{attribute 'linkalways'} 
{attribute 'no_explicit_call' := 'This FB is a CLASS and must be accessed using methods or properties'}
{attribute 'enable_dynamic_creation'}
FUNCTION_BLOCK FINAL MIN_LWORD EXTENDS Node
VAR
	in1 : _LWORD(0);
	in2 : _LWORD(0);
	out : _LWORD(0);
END_VAR

METHOD PUBLIC Clone : I_Node
VAR
	pNode : POINTER TO MIN_LWORD;
END_VAR
pNode := __NEW(MIN_LWORD);
Clone := pNode^;
END_METHOD

METHOD FB_init : BOOL
VAR_INPUT
	bInitRetains : BOOL; // if TRUE, the retain variables are initialized (warm start / cold start)
	bInCopyCode : BOOL;  // if TRUE, the instance afterwards gets moved into the copy code (online change)
END_VAR
AddInput('in1',THIS^.in1);
AddInput('in2',THIS^.in2);
AddOutput('out', THIS^.out);
END_METHOD

METHOD PROTECTED OnExecute
VAR
END_VAR
out.Value := MIN(in1.Value, in2.Value);
END_METHOD

END_FUNCTION_BLOCK

(* stored: Version 1.1.0.1, ProductVersion 3.1.4024.15
   POU MIN_LWORD: Id {a3934d77-3451-408a-9885-6d7c3987b2ac}, SpecialFunc None
   Folder Constructor: Id {6ff46c34-cbba-40a0-be22-35b5975ded58}
   Method Clone: Id {51e5f0d7-02d0-4e01-9958-989d44552127}
   Method FB_init: Id {4cfbed68-a879-483b-88d2-fc73177d910a}
   Method OnExecute: Id {a1b31990-de07-42b4-a0a9-a37781382d8b} *)
